Staubli VAL3: park1.pgx

program park1()
begin
  // -- move back to rest position
  call setSpeed()
  resetMotion()
  movej(jRestPosition, tTool, mFast)
  waitEndMove()
end
